FUNCTION_BLOCK S2_C2 (* Test of sin and cos functions *)
  (* Standard: 61499-1 *)
  (* Version 0.0, 2008-01-16, JHC, Holobloc Inc *)
  (* Compiler header: package fb.rt.student; *)
  (* Compiler classdef: SimpleFB *)
  (* Compiler Java Sun JDK 1.6.0 *)
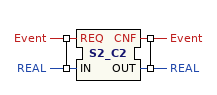
  EVENT_INPUT
    REQ WITH IN; (* Normal Execution Request *)
  END_EVENT
  EVENT_OUTPUT
    CNF WITH OUT; (* Execution Confirmation *)
  END_EVENT
  VAR_INPUT
    IN : REAL;
  END_VAR
  VAR_OUTPUT
    OUT : REAL; (* SIN(IN)**2 + COS(IN)**2, should be 1.0 *)
  END_VAR
  VAR
    SINVAL : REAL;
    COSVAL : REAL;
  END_VAR
  ALGORITHM REQ IN FBD: (* Normally executed algorithm *)
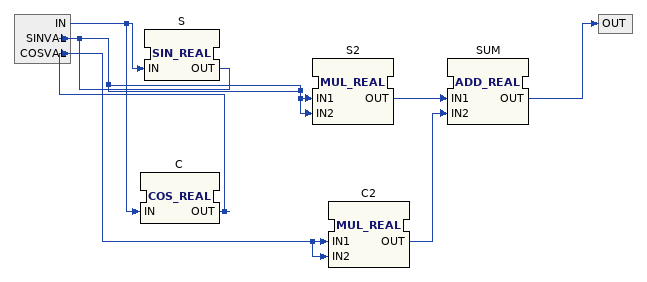
    FBS
      S : SIN_REAL;
      S2 : MUL_REAL;
      C : COS_REAL;
      C2 : MUL_REAL;
      SUM : ADD_REAL;
    END_FBS
    DATA_CONNECTIONS
      IN TO S.IN;
      IN TO C.IN;
      S2.OUT TO SUM.IN1;
      C2.OUT TO SUM.IN2;
      SUM.OUT TO OUT;
      S.OUT TO SINVAL;
      C.OUT TO COSVAL;
      SINVAL TO S2.IN1;
      SINVAL TO S2.IN2;
      COSVAL TO C2.IN1;
      COSVAL TO C2.IN2;
    END_CONNECTIONS
  END_ALGORITHM
END_FUNCTION_BLOCK
